# EPICS alarm handler configuration: Module_8_Alarms_Archiver_Autosave_and_Restore/1_Alarms/ALH-default.alhConfig
GROUP NULL AirCond

GROUP AirCond Temp
CHANNEL Temp ac:odt
CHANNEL Temp ac:idt

GROUP AirCond Power
CHANNEL Power ac:power
